Staubli VAL3: onF5Event.pgx

program onF5Event()
  local string l_sItem
begin
  // look if the bButton is enable
  if bButton[4]
    //
    logMsg("[KERNEL] INTERFACE:PAGE Advance")
  endIf
end
